FUNCTION_BLOCK CompList
VAR_GENERIC CONSTANT
	nCap	: UDINT := 100;
END_VAR

IMPLEMENTS I_MutCompList

VAR
	_iList	: ARRAY[1..nCap] OF I_Component;
	_nLen		: UDINT := 0;
END_VAR

METHOD Append : Result
VAR_INPUT
	iComponent	: I_Component;
	nIndex		: UDINT;
END_VAR
IF nIndex > nCap OR nIndex = 0 THEN
	Append := Err.Ovf;
	RETURN;	
END_IF

IF iComponent = 0 THEN
	IF _iList[nIndex] = 0 THEN
		// Do nothing
		Append := None;
	ELSE
		// Remove
		_iList[nIndex] := 0;
		_nLen := _nLen - 1;
		Append := Ok;
	END_IF
ELSE
	IF _iList[nIndex] = 0 THEN
		// Add
		_iList[nIndex] := iComponent;
		_nLen := _nLen + 1;
		Append := Ok;		
	ELSE
		// Modify
		_iList[nIndex] := iComponent;
		Append := Ok;			
	END_IF
END_IF
END_METHOD

PROPERTY Cap : UDINT
GET
Cap := nCap;
END_GET
END_PROPERTY

METHOD Get : Result
VAR_INPUT
	nIndex		: UDINT;
END_VAR
VAR_OUTPUT
	iComp	: I_Component;
END_VAR
IF _nLen = 0 THEN
	RETURN;
END_IF

IF nIndex > _nLen THEN
	RETURN;
END_IF

IF nIndex > nCap OR_ELSE nIndex < 1 THEN
	Get := Err.Ovf;
	RETURN;
END_IF

iComp := _iList[nIndex];
Get := Ok;
END_METHOD

PROPERTY Length : UDINT
GET
Length := _nLen;
END_GET
END_PROPERTY

END_FUNCTION_BLOCK

(* stored: Version 1.1.0.1
   POU CompList: Id {ca518f37-6c05-4cf4-89d4-75c5e2201c82}, SpecialFunc None
   Method Append: Id {9fb06efd-ab03-4fa1-aa5f-6a55026b07b7}
   Property Cap: Id {50df78aa-587a-44e1-afbf-df9af1ffc7cc}
   Get Get: Id {dfda453b-d7cf-4f39-afd5-c17fcce041a4}
   Method Get: Id {54d36c41-e48b-4d94-a7f2-51e33876950d}
   Property Length: Id {6bac9759-9382-43e1-accb-7021bbfc1551}
   Get Get: Id {464d3f9b-7d83-4738-a4f1-48441410ea69} *)
